SUBAPPLICATION Ventilsteuerung_Uebung_002b (* DigitalInput_I1 auf DigitalOutput_Q1 *)
  (* Standard: 61499-2 *)
  (* Version 1.0, 2023-10-23, franz *)
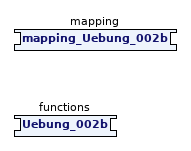
  SUBAPPS
    mapping : mapping_Uebung_002b;
    functions : Uebung_002b;
  END_SUBAPPS
END_SUBAPPLICATION
